// TIA Portal V19 export
TYPE "UDT_MOTORDIRECT"
   STRUCT
      cmd : Struct   // Commands
         auto : Bool := false;
         man : Bool := false;
         start : Bool := false;
         stop : Bool := false;
      END_STRUCT;
      ind : Struct
         auto : Bool := false;
         man : Bool := false;
         start : Bool := false;
         stop : Bool := false;
      END_STRUCT;
      sim : Struct   // Simulation
         fb { S7_SetPoint := 'True'} : Bool := false;   // Feedback simulation
         ctrl { S7_SetPoint := 'True'} : Bool := false;   // Control simulation
      END_STRUCT;
      faults : Struct   // Faults
         ftr { S7_SetPoint := 'True'} : "UDT_ALARMACKN";   // Fail to run
         fts { S7_SetPoint := 'True'} : "UDT_ALARMACKN";   // Fail to stop
         mcb { S7_SetPoint := 'True'} : "UDT_ALARMACKN";   // MCB failure
         ctrl { S7_SetPoint := 'True'} : "UDT_ALARMACKN";   // CTRL failure
         il { S7_SetPoint := 'True'} : "UDT_ALARMACKN";   // Interlock violation
         fpreset : Bool := false;   // Faceplate reset for individual treatment
      END_STRUCT;
      arh : Struct   // Working hours & maintenance timer
         checkafter { S7_SetPoint := 'True'} : DInt := 0;   // Check motor after this SP of working hours
         lastmaint : DInt := 0;   // Last maintenance
         difference : DInt := 0;   // Actual - Last maintenance
         actual : DInt := 0;   // Actual working time (h)
         seconds : DInt := 0;   // seconds counter
         hour : Bool := false;   // 1 hour completed
         resetarh : Bool := false;   // Reset total timer
         enable : Bool := false;   // Enable maintenance
         maintenance : Bool := false;   // Maintenance required
         completed : Bool := false;   // Maintenance completed
      END_STRUCT;
      status : Struct   // Status
         vfb : Bool := false;   // Virtual feedback
         vctrl : Bool := false;   // Virtual control
         ilstart : Bool := false;   // Motor is allowed to start
         fault : Bool := false;   // General fault (generated from the others)
         maint : Bool := false;   // Maintenance required
         icon : Int := 0;
      END_STRUCT;
      delay { S7_SetPoint := 'True'} : "UDT_DELAYONOFF";   // Activation delay on/off
      out : Struct   // Output
         manrun : Bool := false;   // Manual run
         run : Bool := false;   // Command to run
      END_STRUCT;
   END_STRUCT;
END_TYPE
